FUNCTION_BLOCK XtsMover
VAR_INPUT
END_VAR
VAR_OUTPUT
END_VAR
VAR
END_VAR

END_FUNCTION_BLOCK

(* stored: Version 1.1.0.1, ProductVersion 3.1.4024.6
   POU XtsMover: Id {685c76f7-4dc2-4b6a-8a2f-28de7d2e22ba}, SpecialFunc None *)
